FUNCTION F_TimeStamp13_TO_SYSTEMTIME : TimeStruct
VAR_INPUT
	iUnixTimeStamp13 : ULINT;
END_VAR
VAR
	_FileTime64 :T_FILETIME64;
END_VAR

_FileTime64 := (iUnixTimeStamp13 + 11644473600000 - 5000) * 10000;
F_TimeStamp13_TO_SYSTEMTIME := FILETIME64_TO_SYSTEMTIME(_FileTime64);

END_FUNCTION

(* stored: Version 1.1.0.1, ProductVersion 3.1.4024.12
   POU F_TimeStamp13_TO_SYSTEMTIME: Id {e9e8e707-0c6a-4700-b90e-3ec5fabf0760}, SpecialFunc None *)
